PROGRAM INTERNAL P_AdapterExample
VAR
	bStart				: BOOL;
	sValue 				: STRING(255);
	nPos				: T_Size;
	tTime 				: TIME :=  TIME();
	tTime2				: TIME;
	fbStringBuilder 	: FB_StringBuilder;
	fbReadOnlySB 		: FB_ReadOnlyStringBuilderAdapter;
	ipReadOnlySB 		: I_ReadOnlyStringBuilderAdapter;
END_VAR

fbReadOnlySB(ipStringBuilder := fbStringBuilder);
ipReadOnlySB := fbReadOnlySB;

IF bStart THEN
	bStart := FALSE;
	fbStringBuilder
		.Clear()
		.Append('   I love cats.')
		.Append('The time is: ').AppendAny(tTime).Append('.')
		.Append('   ')
		.BTrim();
	END_IF

sValue := ipReadOnlySB
			.Search('T#', 0, Position => nPos)
			.CopySubstringTo(nPos, tc2_Standard.LEN(TIME_TO_STRING(tTime)), tTime2)
			.GetString();

END_PROGRAM

(* stored: Version 1.1.0.1, ProductVersion 3.1.4024.4
   POU P_AdapterExample: Id {c8f6b2a2-2a33-4cec-9fdf-2a33389249e0}, SpecialFunc None *)
